PROGRAM P5_03_OtherControl
VAR
	iSeqControl				:INT;
	tSubStepET				:TIME;
	tSubStepPT				:TIME;
	iSubStepMC				:INT;
	iSubStepPC				:INT;
END_VAR
VAR // added by the converter: edge detectors and wires of the graphical bodies
    _w1, _w2 : TIME;
    _w3, _w4 : BOOL;
END_VAR

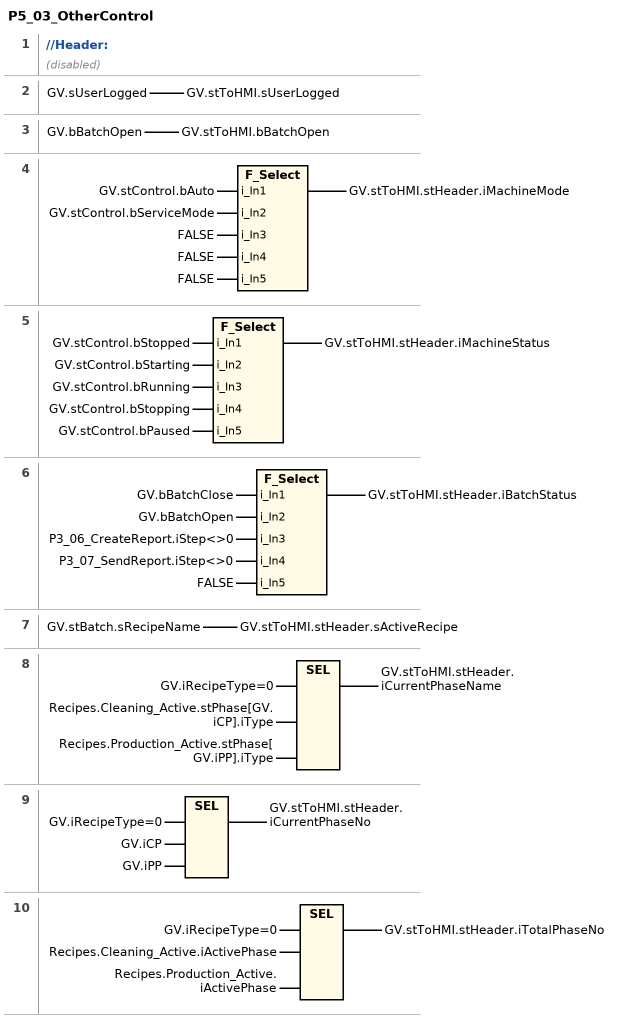
// NETWORK 1 (disabled)
// label: //Header

// NETWORK 2
GV.stToHMI.sUserLogged := GV.sUserLogged;

// NETWORK 3
GV.stToHMI.bBatchOpen := GV.bBatchOpen;

// NETWORK 4
GV.stToHMI.stHeader.iMachineMode := F_Select(i_In1 := GV.stControl.bAuto, i_In2 := GV.stControl.bServiceMode, i_In3 := FALSE, i_In4 := FALSE, i_In5 := FALSE);

// NETWORK 5
GV.stToHMI.stHeader.iMachineStatus := F_Select(i_In1 := GV.stControl.bStopped, i_In2 := GV.stControl.bStarting, i_In3 := GV.stControl.bRunning, i_In4 := GV.stControl.bStopping, i_In5 := GV.stControl.bPaused);

// NETWORK 6
GV.stToHMI.stHeader.iBatchStatus := F_Select(i_In1 := GV.bBatchClose, i_In2 := GV.bBatchOpen, i_In3 := P3_06_CreateReport.iStep<>0, i_In4 := P3_07_SendReport.iStep<>0, i_In5 := FALSE);

// NETWORK 7
GV.stToHMI.stHeader.sActiveRecipe := GV.stBatch.sRecipeName;

// NETWORK 8
GV.stToHMI.stHeader.iCurrentPhaseName := SEL(GV.iRecipeType=0, Recipes.Cleaning_Active.stPhase[GV.iCP].iType, Recipes.Production_Active.stPhase[GV.iPP].iType);

// NETWORK 9
GV.stToHMI.stHeader.iCurrentPhaseNo := SEL(GV.iRecipeType=0, GV.iCP, GV.iPP);

// NETWORK 10
GV.stToHMI.stHeader.iTotalPhaseNo := SEL(GV.iRecipeType=0, Recipes.Cleaning_Active.iActivePhase, Recipes.Production_Active.iActivePhase);

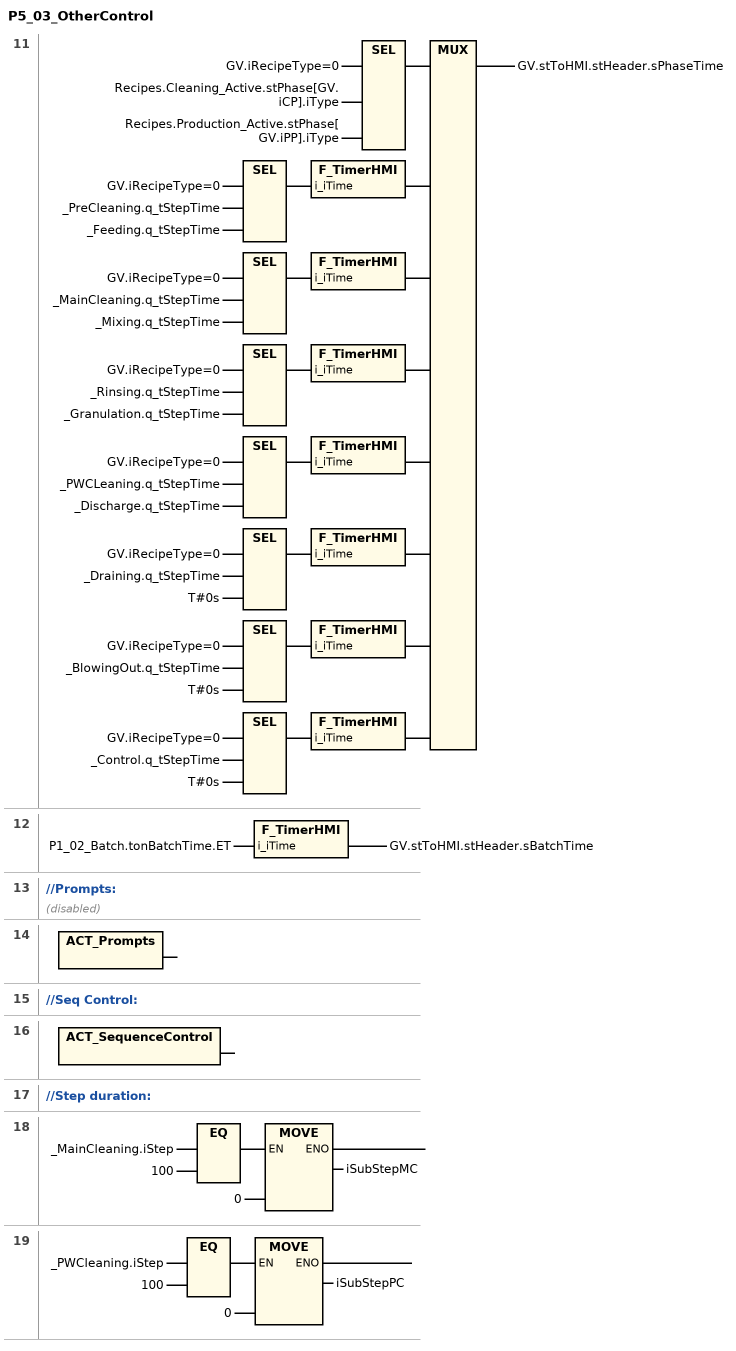
// NETWORK 11
GV.stToHMI.stHeader.sPhaseTime := MUX(SEL(GV.iRecipeType=0, Recipes.Cleaning_Active.stPhase[GV.iCP].iType, Recipes.Production_Active.stPhase[GV.iPP].iType), F_TimerHMI(i_iTime := SEL(GV.iRecipeType=0, _PreCleaning.q_tStepTime, _Feeding.q_tStepTime)), F_TimerHMI(i_iTime := SEL(GV.iRecipeType=0, _MainCleaning.q_tStepTime, _Mixing.q_tStepTime)), F_TimerHMI(i_iTime := SEL(GV.iRecipeType=0, _Rinsing.q_tStepTime, _Granulation.q_tStepTime)), F_TimerHMI(i_iTime := SEL(GV.iRecipeType=0, _PWCLeaning.q_tStepTime, _Discharge.q_tStepTime)), F_TimerHMI(i_iTime := SEL(GV.iRecipeType=0, _Draining.q_tStepTime, T#0s)), F_TimerHMI(i_iTime := SEL(GV.iRecipeType=0, _BlowingOut.q_tStepTime, T#0s)), F_TimerHMI(i_iTime := SEL(GV.iRecipeType=0, _Control.q_tStepTime, T#0s)));

// NETWORK 12
GV.stToHMI.stHeader.sBatchTime := F_TimerHMI(i_iTime := P1_02_Batch.tonBatchTime.ET);

// NETWORK 13 (disabled)
// label: //Prompts

// NETWORK 14
ACT_Prompts();

// NETWORK 15
// label: //Seq Control

// NETWORK 16
ACT_SequenceControl();

// NETWORK 17
// label: //Step duration

// NETWORK 18
IF _MainCleaning.iStep = 100 THEN iSubStepMC := 0; END_IF

// NETWORK 19
IF _PWCleaning.iStep = 100 THEN iSubStepPC := 0; END_IF

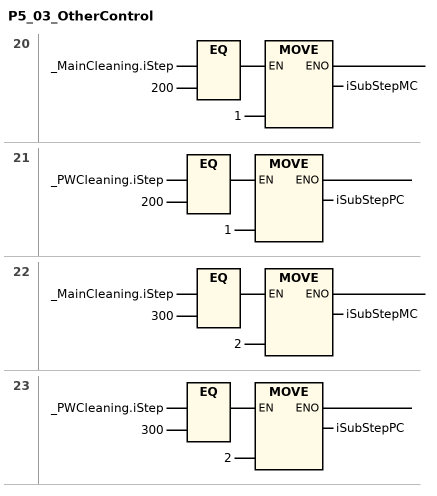
// NETWORK 20
IF _MainCleaning.iStep = 200 THEN iSubStepMC := 1; END_IF

// NETWORK 21
IF _PWCleaning.iStep = 200 THEN iSubStepPC := 1; END_IF

// NETWORK 22
IF _MainCleaning.iStep = 300 THEN iSubStepMC := 2; END_IF

// NETWORK 23
IF _PWCleaning.iStep = 300 THEN iSubStepPC := 2; END_IF

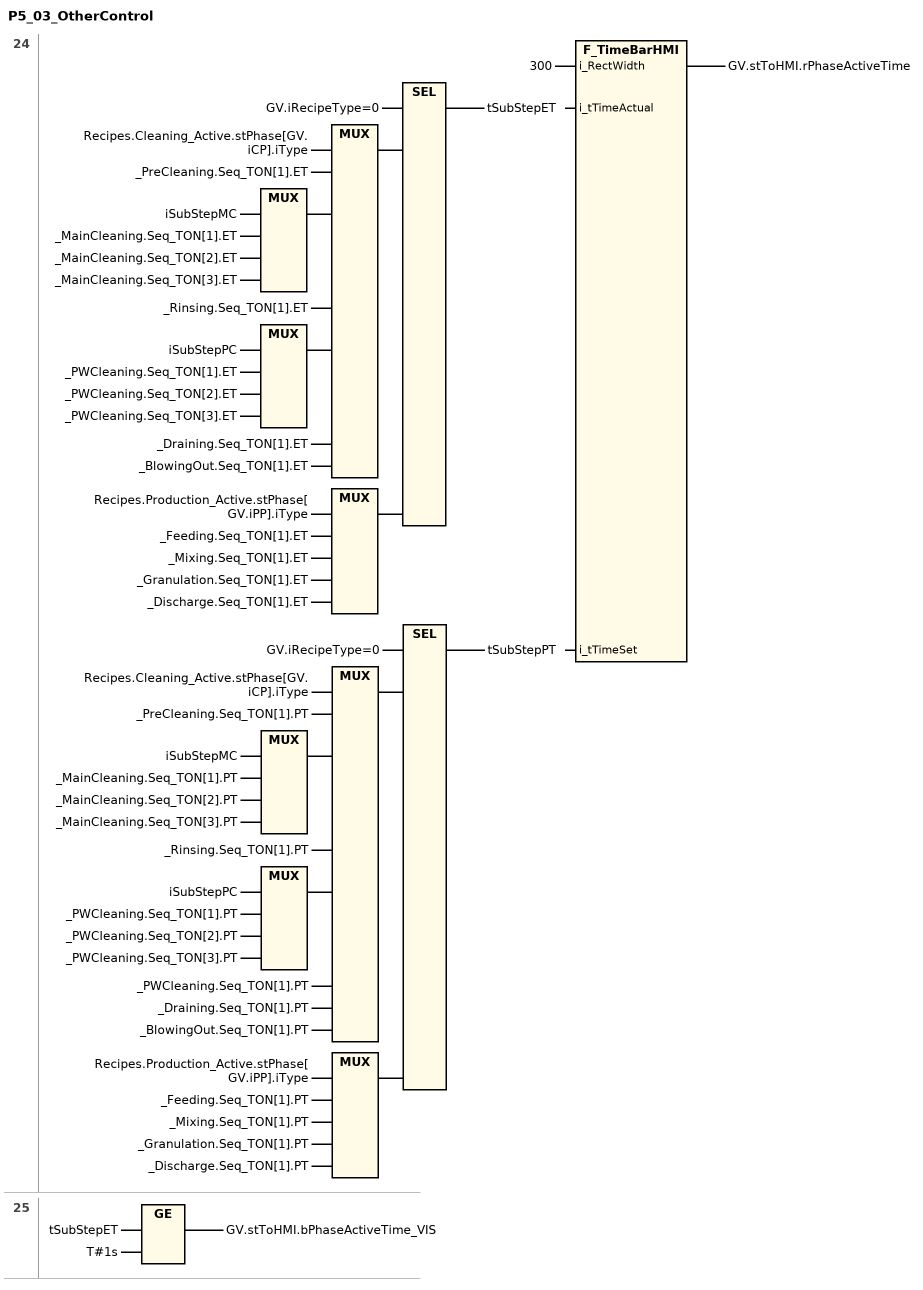
// NETWORK 24
_w1 := SEL(GV.iRecipeType=0, MUX(Recipes.Cleaning_Active.stPhase[GV.iCP].iType, _PreCleaning.Seq_TON[1].ET, MUX(iSubStepMC, _MainCleaning.Seq_TON[1].ET, _MainCleaning.Seq_TON[2].ET, _MainCleaning.Seq_TON[3].ET), _Rinsing.Seq_TON[1].ET, MUX(iSubStepPC, _PWCleaning.Seq_TON[1].ET, _PWCleaning.Seq_TON[2].ET, _PWCleaning.Seq_TON[3].ET), _Draining.Seq_TON[1].ET, _BlowingOut.Seq_TON[1].ET), MUX(Recipes.Production_Active.stPhase[GV.iPP].iType, _Feeding.Seq_TON[1].ET, _Mixing.Seq_TON[1].ET, _Granulation.Seq_TON[1].ET, _Discharge.Seq_TON[1].ET));
tSubStepET := _w1;
_w2 := SEL(GV.iRecipeType=0, MUX(Recipes.Cleaning_Active.stPhase[GV.iCP].iType, _PreCleaning.Seq_TON[1].PT, MUX(iSubStepMC, _MainCleaning.Seq_TON[1].PT, _MainCleaning.Seq_TON[2].PT, _MainCleaning.Seq_TON[3].PT), _Rinsing.Seq_TON[1].PT, MUX(iSubStepPC, _PWCleaning.Seq_TON[1].PT, _PWCleaning.Seq_TON[2].PT, _PWCleaning.Seq_TON[3].PT), _PWCleaning.Seq_TON[1].PT, _Draining.Seq_TON[1].PT, _BlowingOut.Seq_TON[1].PT), MUX(Recipes.Production_Active.stPhase[GV.iPP].iType, _Feeding.Seq_TON[1].PT, _Mixing.Seq_TON[1].PT, _Granulation.Seq_TON[1].PT, _Discharge.Seq_TON[1].PT));
tSubStepPT := _w2;
GV.stToHMI.rPhaseActiveTime := F_TimeBarHMI(i_RectWidth := 300, i_tTimeActual := _w1, i_tTimeSet := _w2);

// NETWORK 25
GV.stToHMI.bPhaseActiveTime_VIS := tSubStepET >= T#1s;

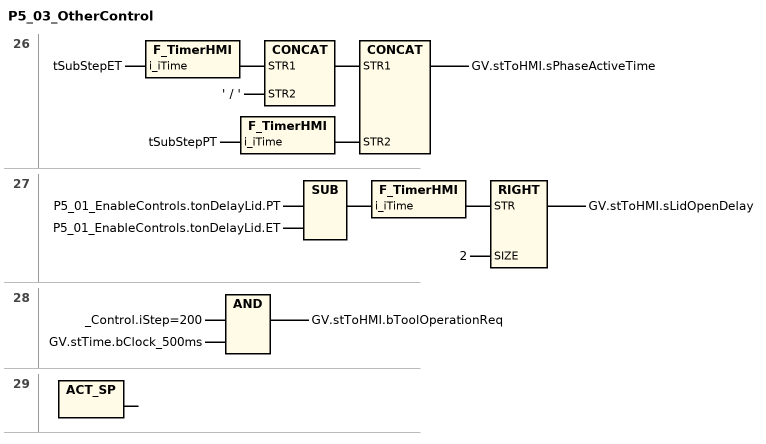
// NETWORK 26
GV.stToHMI.sPhaseActiveTime := CONCAT(STR1 := CONCAT(STR1 := F_TimerHMI(i_iTime := tSubStepET), STR2 := ' / '), STR2 := F_TimerHMI(i_iTime := tSubStepPT));

// NETWORK 27
GV.stToHMI.sLidOpenDelay := RIGHT(STR := F_TimerHMI(i_iTime := P5_01_EnableControls.tonDelayLid.PT - P5_01_EnableControls.tonDelayLid.ET), SIZE := 2);

// NETWORK 28
GV.stToHMI.bToolOperationReq := (_Control.iStep=200) AND GV.stTime.bClock_500ms;

// NETWORK 29
ACT_SP();

ACTION ACT_Prompts:
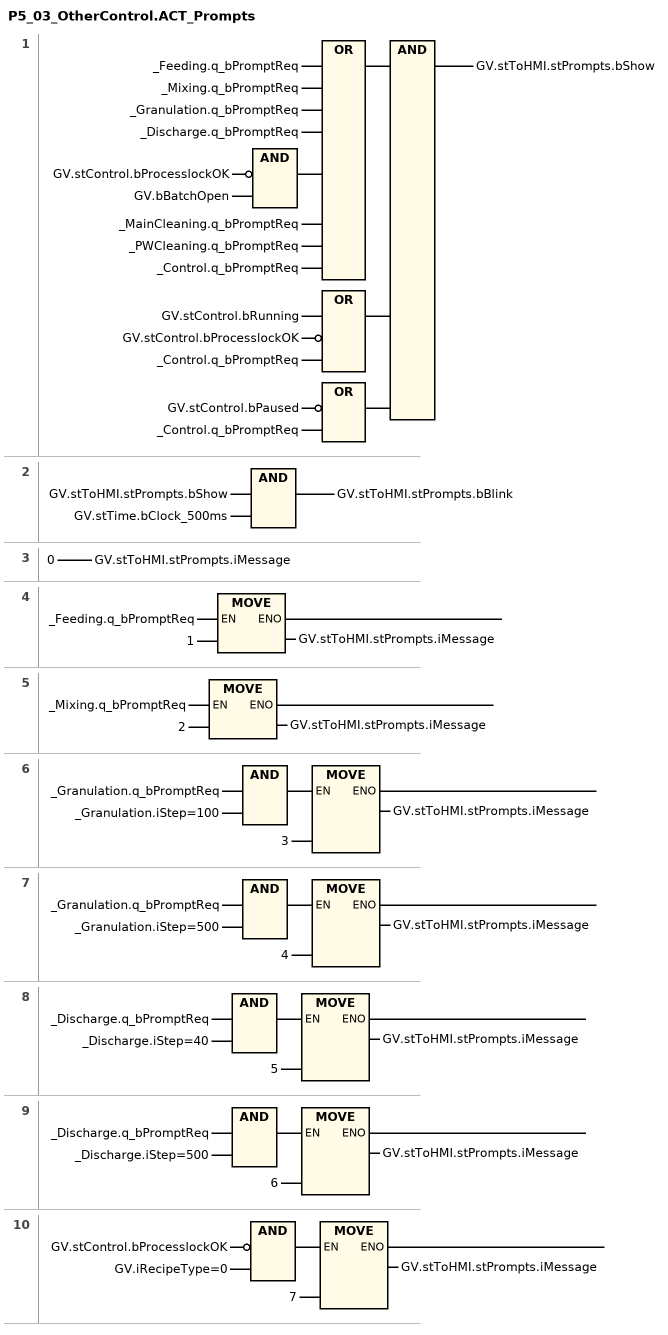
// NETWORK 1
GV.stToHMI.stPrompts.bShow := (_Feeding.q_bPromptReq OR _Mixing.q_bPromptReq OR _Granulation.q_bPromptReq OR _Discharge.q_bPromptReq OR NOT GV.stControl.bProcesslockOK AND GV.bBatchOpen OR _MainCleaning.q_bPromptReq OR _PWCleaning.q_bPromptReq OR _Control.q_bPromptReq) AND (GV.stControl.bRunning OR NOT GV.stControl.bProcesslockOK OR _Control.q_bPromptReq) AND (NOT GV.stControl.bPaused OR _Control.q_bPromptReq);

// NETWORK 2
GV.stToHMI.stPrompts.bBlink := GV.stToHMI.stPrompts.bShow AND GV.stTime.bClock_500ms;

// NETWORK 3
GV.stToHMI.stPrompts.iMessage := 0;

// NETWORK 4
IF _Feeding.q_bPromptReq THEN GV.stToHMI.stPrompts.iMessage := 1; END_IF

// NETWORK 5
IF _Mixing.q_bPromptReq THEN GV.stToHMI.stPrompts.iMessage := 2; END_IF

// NETWORK 6
IF _Granulation.q_bPromptReq AND (_Granulation.iStep=100) THEN GV.stToHMI.stPrompts.iMessage := 3; END_IF

// NETWORK 7
IF _Granulation.q_bPromptReq AND (_Granulation.iStep=500) THEN GV.stToHMI.stPrompts.iMessage := 4; END_IF

// NETWORK 8
IF _Discharge.q_bPromptReq AND (_Discharge.iStep=40) THEN GV.stToHMI.stPrompts.iMessage := 5; END_IF

// NETWORK 9
IF _Discharge.q_bPromptReq AND (_Discharge.iStep=500) THEN GV.stToHMI.stPrompts.iMessage := 6; END_IF

// NETWORK 10
IF NOT GV.stControl.bProcesslockOK AND (GV.iRecipeType=0) THEN GV.stToHMI.stPrompts.iMessage := 7; END_IF

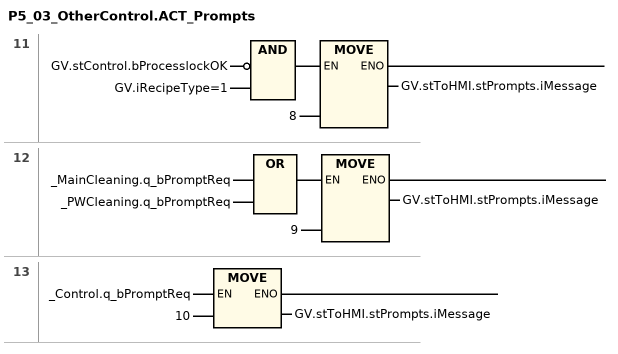
// NETWORK 11
IF NOT GV.stControl.bProcesslockOK AND (GV.iRecipeType=1) THEN GV.stToHMI.stPrompts.iMessage := 8; END_IF

// NETWORK 12
IF _MainCleaning.q_bPromptReq OR _PWCleaning.q_bPromptReq THEN GV.stToHMI.stPrompts.iMessage := 9; END_IF

// NETWORK 13
IF _Control.q_bPromptReq THEN GV.stToHMI.stPrompts.iMessage := 10; END_IF
END_ACTION

ACTION ACT_SequenceControl:
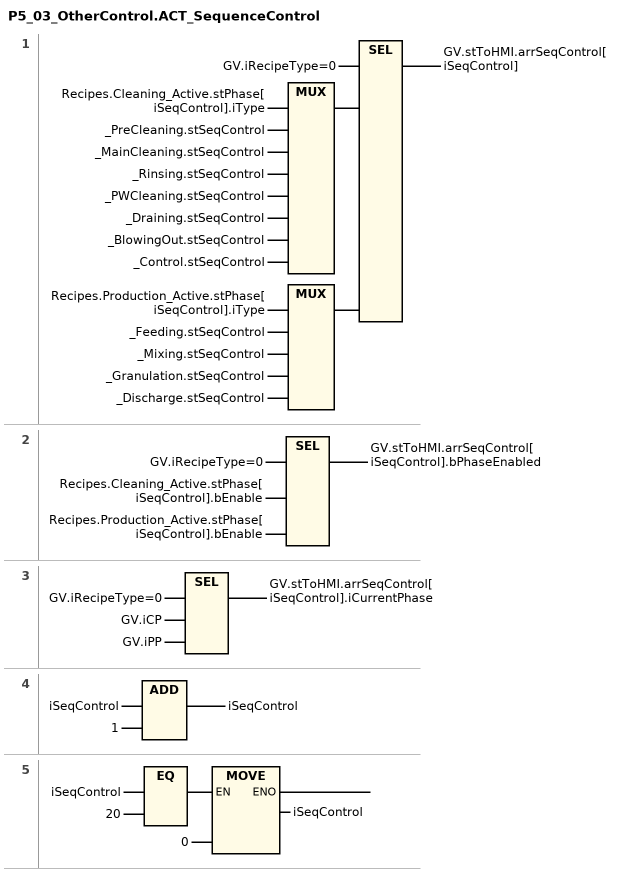
// NETWORK 1
GV.stToHMI.arrSeqControl[iSeqControl] := SEL(GV.iRecipeType=0, MUX(Recipes.Cleaning_Active.stPhase[iSeqControl].iType, _PreCleaning.stSeqControl, _MainCleaning.stSeqControl, _Rinsing.stSeqControl, _PWCleaning.stSeqControl, _Draining.stSeqControl, _BlowingOut.stSeqControl, _Control.stSeqControl), MUX(Recipes.Production_Active.stPhase[iSeqControl].iType, _Feeding.stSeqControl, _Mixing.stSeqControl, _Granulation.stSeqControl, _Discharge.stSeqControl));

// NETWORK 2
GV.stToHMI.arrSeqControl[iSeqControl].bPhaseEnabled := SEL(GV.iRecipeType=0, Recipes.Cleaning_Active.stPhase[iSeqControl].bEnable, Recipes.Production_Active.stPhase[iSeqControl].bEnable);

// NETWORK 3
GV.stToHMI.arrSeqControl[iSeqControl].iCurrentPhase := SEL(GV.iRecipeType=0, GV.iCP, GV.iPP);

// NETWORK 4
iSeqControl := iSeqControl + 1;

// NETWORK 5
IF iSeqControl = 20 THEN iSeqControl := 0; END_IF
END_ACTION

ACTION ACT_SP:
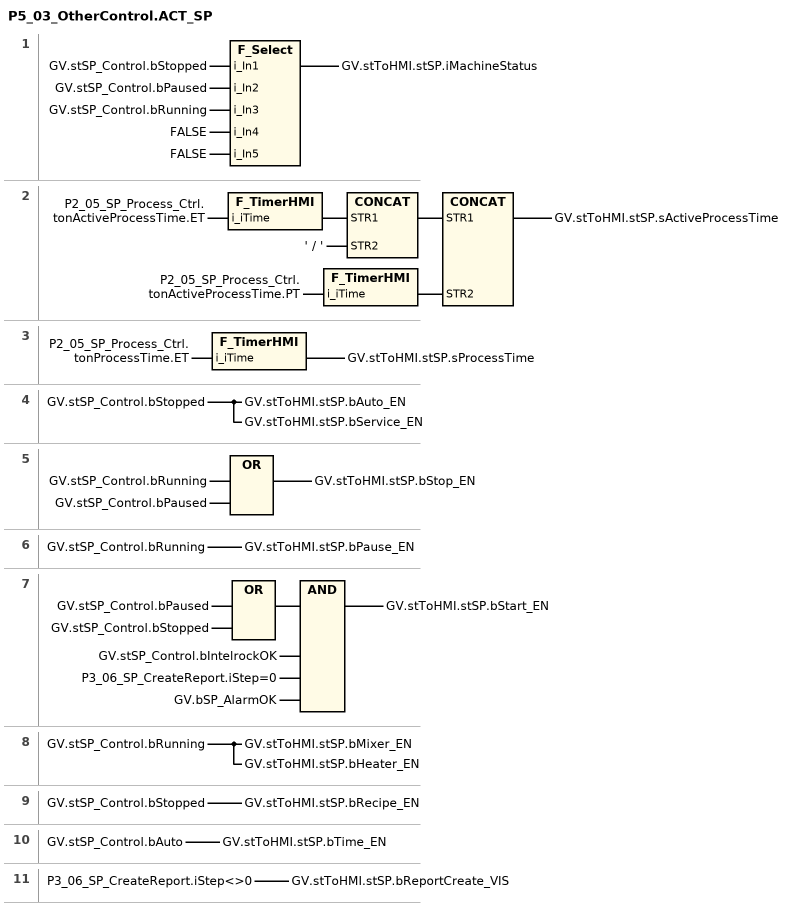
// NETWORK 1
GV.stToHMI.stSP.iMachineStatus := F_Select(i_In1 := GV.stSP_Control.bStopped, i_In2 := GV.stSP_Control.bPaused, i_In3 := GV.stSP_Control.bRunning, i_In4 := FALSE, i_In5 := FALSE);

// NETWORK 2
GV.stToHMI.stSP.sActiveProcessTime := CONCAT(STR1 := CONCAT(STR1 := F_TimerHMI(i_iTime := P2_05_SP_Process_Ctrl.tonActiveProcessTime.ET), STR2 := ' / '), STR2 := F_TimerHMI(i_iTime := P2_05_SP_Process_Ctrl.tonActiveProcessTime.PT));

// NETWORK 3
GV.stToHMI.stSP.sProcessTime := F_TimerHMI(i_iTime := P2_05_SP_Process_Ctrl.tonProcessTime.ET);

// NETWORK 4
_w3 := GV.stSP_Control.bStopped;
GV.stToHMI.stSP.bAuto_EN := _w3;
GV.stToHMI.stSP.bService_EN := _w3;

// NETWORK 5
GV.stToHMI.stSP.bStop_EN := GV.stSP_Control.bRunning OR GV.stSP_Control.bPaused;

// NETWORK 6
GV.stToHMI.stSP.bPause_EN := GV.stSP_Control.bRunning;

// NETWORK 7
GV.stToHMI.stSP.bStart_EN := (GV.stSP_Control.bPaused OR GV.stSP_Control.bStopped) AND GV.stSP_Control.bIntelrockOK AND (P3_06_SP_CreateReport.iStep=0) AND GV.bSP_AlarmOK;

// NETWORK 8
_w4 := GV.stSP_Control.bRunning;
GV.stToHMI.stSP.bMixer_EN := _w4;
GV.stToHMI.stSP.bHeater_EN := _w4;

// NETWORK 9
GV.stToHMI.stSP.bRecipe_EN := GV.stSP_Control.bStopped;

// NETWORK 10
GV.stToHMI.stSP.bTime_EN := GV.stSP_Control.bAuto;

// NETWORK 11
GV.stToHMI.stSP.bReportCreate_VIS := P3_06_SP_CreateReport.iStep<>0;
END_ACTION

END_PROGRAM

(* stored: Version 1.1.0.1, ProductVersion 3.1.4026.13
   POU P5_03_OtherControl: Id {3767f6b8-37b7-4d6c-944a-65dae6712b2d}, SpecialFunc None
   Action ACT_Prompts: Id {0878575b-1350-42bb-86c8-d1d075c4f1a4}
   Action ACT_SequenceControl: Id {8879beec-4859-4407-8077-14ace9c1a8c7}
   Action ACT_SP: Id {02d1ec0c-7e85-4007-b0bf-3d00be1cee2a} *)
